TYPE ST_CoolingSystem_Get :
STRUCT
	CoolingSystemMode		:	eCoolingSystemState;
	HeatPumpStatus			: 	eHeatPumpState;
	r_CoolantTemperature	:	REAL;
	r_CoolantPressure		:	REAL;
	r_EnclosureDewpoint		:	REAL;
	ui_DehumRemainingTime	: 	UINT; //minutes
		
	
	HeatPumpSystem 			: REFERENCE TO ST_HeatpumpSystemGet;	
	Events					: ST_CoolingSystem_Events;
END_STRUCT
END_TYPE

(* stored: Version 1.1.0.1, ProductVersion 3.1.4024.12
   DUT ST_CoolingSystem_Get: Id {c5f9e8e4-f620-4cbc-bb65-ad5a08f7db42} *)
